{attribute 'pack_mode' := '1'}
TYPE ST_MsgToPLC EXTENDS ST_PLCMsg:
STRUCT
    lowUUID		: LINT;	(* The low-order part of the UUID. *)
    highUUID	: LINT;	(* The high-order part of the UUID. *)
    dtime		: DINT;	(* Time of day of sending, in milliseconds. *)
    sequence	: DINT := 1;	(* Message sequence number. *)
END_STRUCT
END_TYPE

(* stored: Version 1.1.0.1, ProductVersion 3.1.4022.18
   DUT ST_MsgToPLC: Id {987d0f11-b4fb-4391-86af-0a6bd82a8e9f} *)
